// SIMATIC S7-200 project (STEP 7-Micro/WIN), CPU 224XP CN REL 02.01

ORGANIZATION_BLOCK 主程序:OB1
TITLE=程序注释
BEGIN
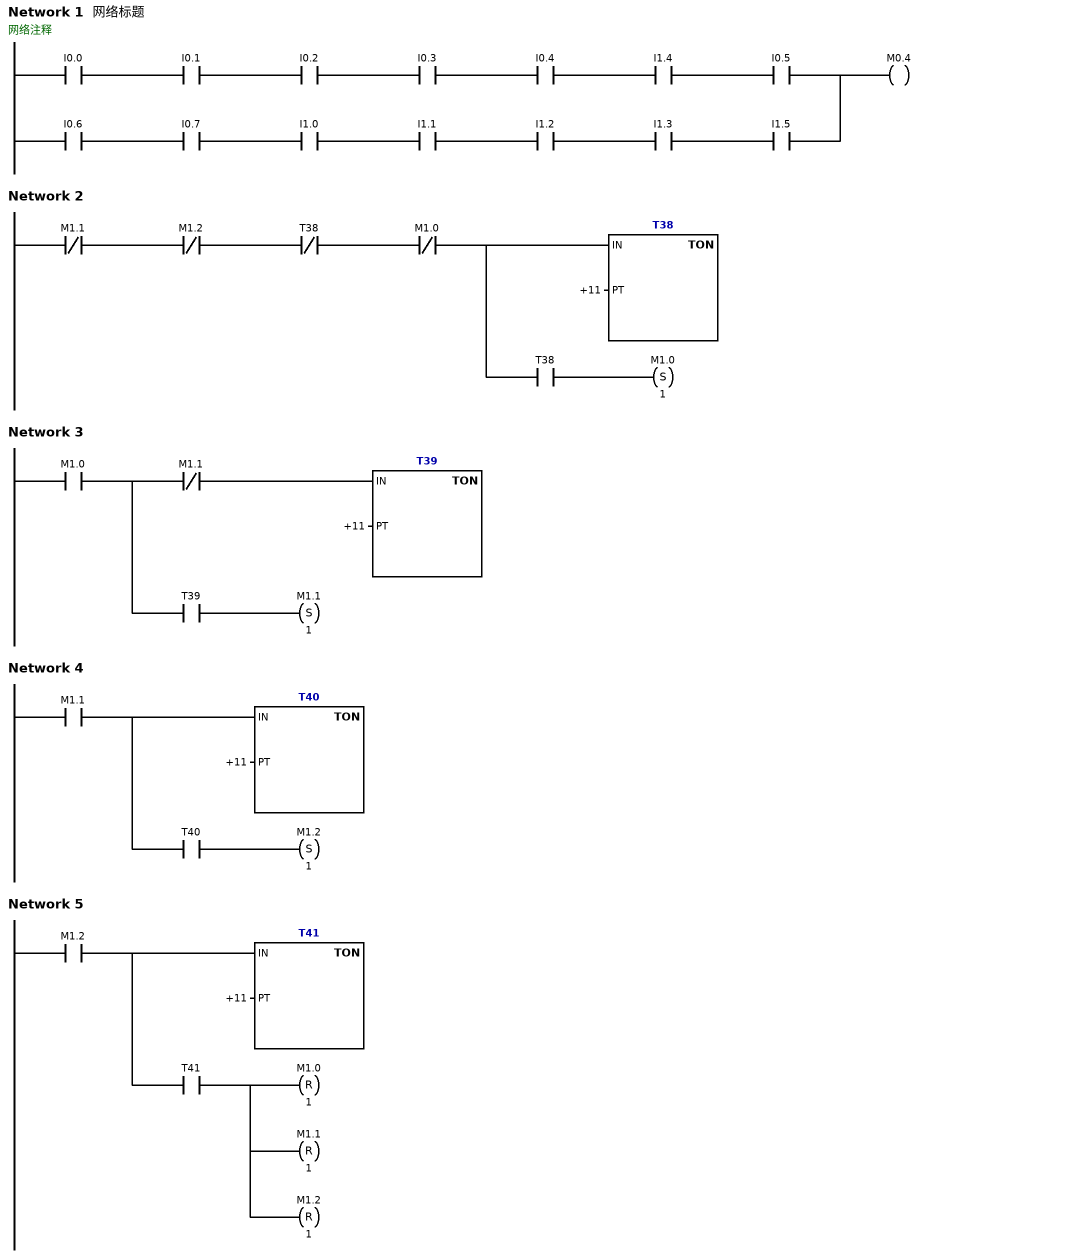
Network 1 // 网络标题
// 网络注释
LD     I0.0
A      I0.1
A      I0.2
A      I0.3
A      I0.4
A      I1.4
A      I0.5
LD     I0.6
A      I0.7
A      I1.0
A      I1.1
A      I1.2
A      I1.3
A      I1.5
OLD
=      M0.4
Network 2
LDN    M1.1
AN     M1.2
AN     T38
AN     M1.0
TON    T38, +11
A      T38
S      M1.0, 1
Network 3
LD     M1.0
LPS
AN     M1.1
TON    T39, +11
LPP
A      T39
S      M1.1, 1
Network 4
LD     M1.1
TON    T40, +11
A      T40
S      M1.2, 1
Network 5
LD     M1.2
TON    T41, +11
A      T41
R      M1.0, 1
R      M1.1, 1
R      M1.2, 1
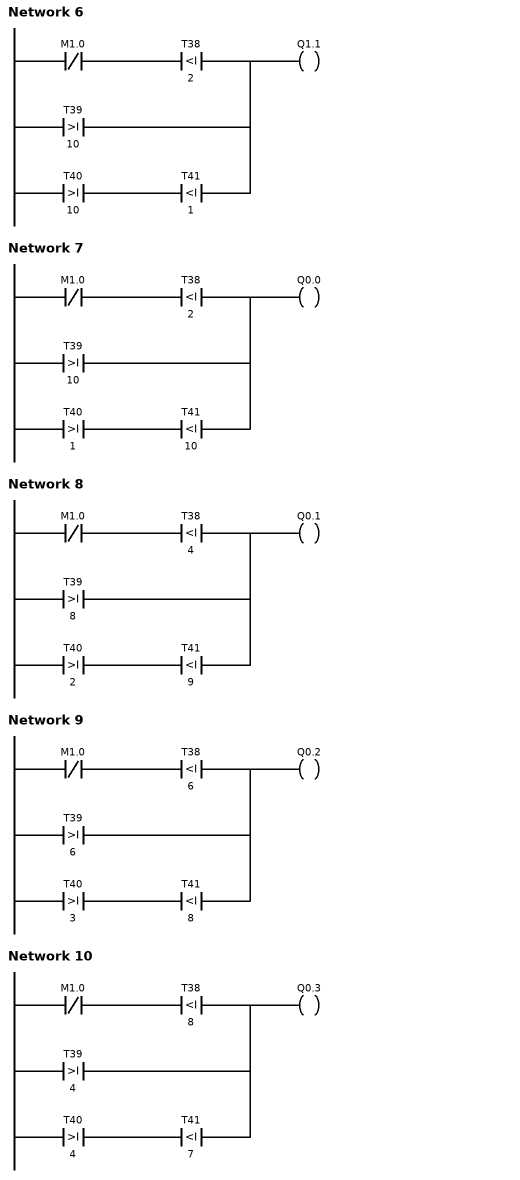
Network 6
LDN    M1.0
AW<    T38, 2
OW>    T39, 10
LDW>   T40, 10
AW<    T41, 1
OLD
=      Q1.1
Network 7
LDN    M1.0
AW<    T38, 2
OW>    T39, 10
LDW>   T40, 1
AW<    T41, 10
OLD
=      Q0.0
Network 8
LDN    M1.0
AW<    T38, 4
OW>    T39, 8
LDW>   T40, 2
AW<    T41, 9
OLD
=      Q0.1
Network 9
LDN    M1.0
AW<    T38, 6
OW>    T39, 6
LDW>   T40, 3
AW<    T41, 8
OLD
=      Q0.2
Network 10
LDN    M1.0
AW<    T38, 8
OW>    T39, 4
LDW>   T40, 4
AW<    T41, 7
OLD
=      Q0.3
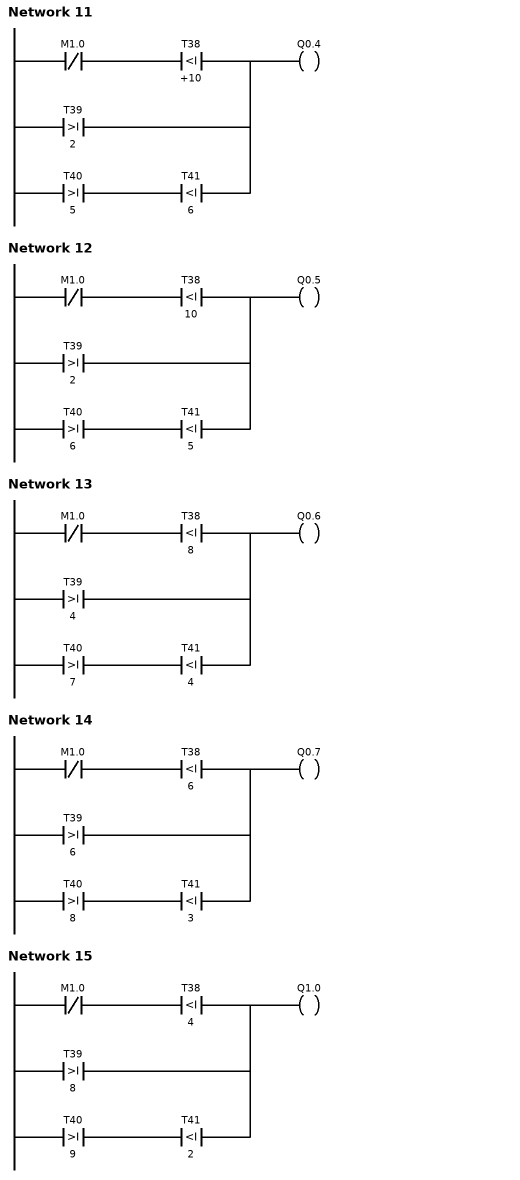
Network 11
LDN    M1.0
AW<    T38, +10
OW>    T39, 2
LDW>   T40, 5
AW<    T41, 6
OLD
=      Q0.4
Network 12
LDN    M1.0
AW<    T38, 10
OW>    T39, 2
LDW>   T40, 6
AW<    T41, 5
OLD
=      Q0.5
Network 13
LDN    M1.0
AW<    T38, 8
OW>    T39, 4
LDW>   T40, 7
AW<    T41, 4
OLD
=      Q0.6
Network 14
LDN    M1.0
AW<    T38, 6
OW>    T39, 6
LDW>   T40, 8
AW<    T41, 3
OLD
=      Q0.7
Network 15
LDN    M1.0
AW<    T38, 4
OW>    T39, 8
LDW>   T40, 9
AW<    T41, 2
OLD
=      Q1.0
END_ORGANIZATION_BLOCK
